(****************************************************************************************)
(*							Beckhoff Automation Poland									*)
(*							GRAYW_TO_WORD	 v1.0										*)
(*									29.12.2008											*)
(*		Funkcja konwerująca wartosc wejsciowa typu WORD zapisana w kodzie Graya			*)
(*						 na wartosc decymalna typu WORD									*)
(*______________________________________________________________________________________*)
FUNCTION GRAYW_TO_WORD : WORD
VAR_INPUT
	wIn:WORD;
END_VAR
VAR
END_VAR

GRAYW_TO_WORD.15 := wIn.15 XOR 0;
GRAYW_TO_WORD.14 := wIn.14 XOR GRAYW_TO_WORD.15;
GRAYW_TO_WORD.13 := wIn.13 XOR GRAYW_TO_WORD.14;
GRAYW_TO_WORD.12 := wIn.12 XOR GRAYW_TO_WORD.13;
GRAYW_TO_WORD.11 := wIn.11 XOR GRAYW_TO_WORD.12;
GRAYW_TO_WORD.10 := wIn.10 XOR GRAYW_TO_WORD.11;
GRAYW_TO_WORD.9 := wIn.9 XOR GRAYW_TO_WORD.10;
GRAYW_TO_WORD.8 := wIn.8 XOR GRAYW_TO_WORD.9;
GRAYW_TO_WORD.7 := wIn.7 XOR GRAYW_TO_WORD.8;
GRAYW_TO_WORD.6 := wIn.6 XOR GRAYW_TO_WORD.7;
GRAYW_TO_WORD.5 := wIn.5 XOR GRAYW_TO_WORD.6;
GRAYW_TO_WORD.4 := wIn.4 XOR GRAYW_TO_WORD.5;
GRAYW_TO_WORD.3 := wIn.3 XOR GRAYW_TO_WORD.4;
GRAYW_TO_WORD.2 := wIn.2 XOR GRAYW_TO_WORD.3;
GRAYW_TO_WORD.1 := wIn.1 XOR GRAYW_TO_WORD.2;
GRAYW_TO_WORD.0 := wIn.0 XOR GRAYW_TO_WORD.1;

END_FUNCTION

(* stored: Version 1.1.0.1, ProductVersion 3.1.4026.13, FileIdentifier 08ec6c88294cc854553fb47f8a933e97b1963487, FileSignature 15091294911cbb8cb8580a3f5e6e7afbcf997dfafe72a8b2804a7329173e9b3861e469d08f5276daef59dadc95f0098795570d931fbaea7bb6ca6a848a6c45326b7ce584f9f8bcc276601b31c50edb60094456a89d5c6ad23b39c964da350c1e7c28cf9a63299b30e0944eeef057c74cd6a01b59404b6f7bbe34c21f7d41120eb1c09ab02fe40a6f7cd312a4b7f3741915ea6f539b2ebfbe5b194c5648bfd20507e60320cac8b3827db7b3f8ec0f94cf8bab35120f61d500f844aeb9c8cda1e50e7b8232510c9f5765a62c173ff893be94c7cc2ff8313f73fd34570fb417f895b2d2a0b5c6b7d44146096b6ea7aa8f9716052b599559734a027c1b4bae6bb03e
   POU GRAYW_TO_WORD: Id {18ed0d3f-424d-46cf-8b12-fcb1fd2aa7c2}, SpecialFunc None *)
